FUNCTION_BLOCK FB_GeneratorEx EXTENDS FB_Generator
VAR_INPUT
END_VAR
VAR_OUTPUT
END_VAR
VAR
END_VAR

{warning 'add method implementation'}
METHOD Flash : BOOL
ton1(IN:=NOT ton1.Q , PT:= tCycleTime, Q=> , ET=> );



// duty ratio 33% ON, 67% Off

Flash := ton1.ET < ton1.PT/3;
END_METHOD

PROPERTY P_tCycleTime : TIME
GET
P_tCycleTime := tCycleTime;
END_GET
SET
IF P_tCycleTime < T#50MS THEN 
	tCycleTime := T#50MS;
ELSIF P_tCycleTime > T#5S THEN 
	tCycleTime := T#5S;
ELSE
	tCycleTime := P_tCycleTime;	
END_IF
END_SET
END_PROPERTY

PROPERTY P_Vendor : STRING
GET
P_Vendor := CONCAT('MicroSoft',SUPER^.P_Vendor);
END_GET
END_PROPERTY

END_FUNCTION_BLOCK

(* stored: Version 1.1.0.1, ProductVersion 3.1.4022.16
   POU FB_GeneratorEx: Id {87f842f4-f1dd-4c6d-bc76-6b91d07682bc}, SpecialFunc None
   Method Flash: Id {4d06014e-db69-44ce-adb5-e718c95b7108}
   Property P_tCycleTime: Id {fc5cc02e-2a69-43d2-aea5-fe196018c2bb}
   Get Get: Id {1e50ad76-4661-4a6d-b2b8-8fac3c819521}
   Set Set: Id {39e907be-68b4-4327-9f9c-6ccd6355ad8a}
   Property P_Vendor: Id {d1d7dd62-6965-43e6-a38e-76772b481be1}
   Get Get: Id {939de465-8ae0-43a0-a09a-faa0834988d4} *)
